{attribute 'qualified_only'}
VAR_GLOBAL CONSTANT
    nDefaultCapacity: UDINT := 4;
    nMaxLength: UDINT := 16#7FEFFFFF;
END_VAR

(* stored: Version 1.1.0.1, ProductVersion 3.1.4024.12
   GVL Param_List: Id {317121e1-9a4d-09e4-2c0b-5ad0a839b269}, ParameterList True *)
